{attribute 'GeneratedUsingTerminal: DL-EC1A-0000'}
{attribute addProperty BoxType "DL-EC1A-0000"}
{attribute addProperty Id "Tool_01_ScoreAT %I*DINT4"}
{attribute addProperty CRC "2706247979"}
{attribute addProperty Size "4"}
TYPE ID03_Current_Value_A14E112B EXTENDS InputBase_8311D824 :
STRUCT
	{attribute addProperty Name "Tool_01_Score"}
	Tool_01_Score AT %I* : DINT;
END_STRUCT
END_TYPE

(* stored: Version 1.1.0.1, ProductVersion 3.1.4024.12
   DUT ID03_Current_Value_A14E112B: Id {2b7294cb-9bd6-0bd0-0fa0-636787c8ce4a} *)
